                       // Move received data to output
                       #tempRet := INT_TO_WORD(MOVE_BLK_VARIANT(SRC := #statRcvBuffer,
                                                                                        COUNT := MIN(IN1 := #tempChunk.lenData, IN2 := #statSizeRcvArray - #statRcvdLen), // Move as much as possible to output
                                                                                        SRC_INDEX := #tempChunk.posData,
                                                                                        DEST_INDEX := UDINT_TO_DINT(#statRcvdLen),
                                                                                        DEST => #responseData));

                       // Exit loop immediately and output error if data could not be moved
                       IF #tempRet <> 0 THEN
                         #statStatusID := #STATUS_ID_MOVE_CHUNKED;
                         #statStatus := #tempRet;
                         EXIT;
                       END_IF;

                       // Move start position of data behind data of current chunk in case packet contains more data; only relevant if REPEAT loop is executed again
                       #tempChunk.posData += #tempChunk.lenData;

                       // Subtract length of data in current packet from remaining length of chunk and add to sum of received data
                       #statChunkLen -= #tempChunk.lenData;
                       #statRcvdLen += #tempChunk.lenData;

                       IF #statRcvdLen > #statSizeRcvArray THEN // Receive buffer too small
                         #statStatus := #STATUS_BUFFER_SIZE;
                         #statLength := #statRcvdLen; // Output required size of buffer according to so far received chunked messages
                       END_IF;
                     END_IF;
                   UNTIL (#tempChunk.exitLoop = true) END_REPEAT;
                 END_IF;
               END_REGION

             ELSIF #instTRcv.ERROR THEN
               #statStatusID := #STATUS_ID_TRCV;
               #statStatus := #instTRcv.STATUS;
             END_IF;
           END_REGION

         ELSE // Undefined state in state machine reached
           #statStatus := #STATUS_UNDEFINED_STATE;
       END_CASE;

     UNTIL (#tempExitLoop = true) END_REPEAT;
   END_REGION

   REGION OUTPUTS
     // Write outputs
     IF (#statStatus = #STATUS_DONE) AND (#statDone = false) THEN // Execution finished without errors
       #statDone := true;
       #statBusy := false;
       #statError := false;
       #statSend.connect := false;
       #statSend.req := false;
       #statTimeoutIn := false;
       #statFBState := #STATE_IDLE; // Switch state machine to "no processing"

     ELSIF (#statStatus.%X15 = true) AND (#statError = false) THEN // Error occurred (#statStatus is 16#8000 to 16#FFFF)
       #statDone := false;
       #statBusy := false;
       #statError := true;
       #statSend.connect := false;
       #statSend.req := false;
       #statTimeoutIn := false;
       #statFBState := #STATE_IDLE; // Switch state machine to "no processing"

     ELSIF (#execute = false) AND ((#statDone = true) OR (#statError = true)) THEN // Reset outputs
       #statDone := false;
       #statBusy := false;
       #statError := false;
       #statStatusID := 0;
       #statStatus := #STATUS_IDLE;
       #statResponseCode := 0;
       #statLength := 0;
       #statContentLength := 0;
       #statChunkLen := 0;
       #statEncoding := '';
       #statRcvdLen := 0;
       #statTimeoutIn := false;
     END_IF;

     // Write static values to outputs
     #done := #statDone;
     #busy := #statBusy;
     #error := #statError;
     #statusID := #statStatusID;
     #status := #statStatus;
     #responseCode := #statResponseCode;
     #length := #statLength;
   END_REGION OUTPUTS
END_FUNCTION_BLOCK

// folder: REST/Utilities

FUNCTION "LHTTP_ExtractStringFromArray" : Word   // FC2, SCL
{ S7_Optimized_Access := 'TRUE' }
VERSION : 0.1
   VAR_INPUT
      textBefore : String;   // Text before text that is extracted
      textAfter : String;   // Text after text that is extracted
   END_VAR
   VAR_OUTPUT
      extractedString : String;   // Extracted string
   END_VAR
   VAR_IN_OUT
      searchIn : Array[*] of Char;   // Array of Char to search in
   END_VAR
   VAR_TEMP
      tempLowerBound : DInt;   // Lower bound of given array
      tempNumElements : UDInt;   // Number of elements in given array
      tempPosInArray : DInt;   // Position in array during search
      tempLenTextBefore : Int;   // Length of text before
      tempPosTextBefore : DInt;   // Position of text before in array of Char
      tempLenTextAfter : Int;   // Length of text after
      tempPosTextAfter : Int;   // Position of text after in converted string
      tempString : String;   // Temporary string to work with
   END_VAR
   // Ret_Val : Return value; 16#0000: Successful, text was found, 16#9001: Unsuccessful, only start text was found, extracted String is filled with characters after start text, 16#9002: Unsuccessful, neither text was found
   VAR CONSTANT
      LEN_STRING : UInt := 254;   // Max. length of String
      STATUS_TEXT_FOUND : Word := 16#0000;   // Texts before and after were found
      STATUS_ONLY_START : Word := 16#9001;   // Only text before was found
      STATUS_NOTHING_FOUND : Word := 16#9002;   // Neither text was found
   END_VAR
BEGIN
   //=============================================================================
   // SIEMENS AG
   // (c)Copyright 2019
   //-----------------------------------------------------------------------------
   // Library:       LHTTP
   // Tested with:   CPU 1516-3 PN/DP V2.6
   // Engineering:   TIA Portal V15.1
   // Restrictions:  --
   // Requirements:  --
   // Functionality: Extracts a String specified by a text before and after
   //                from an array of Char
   //-----------------------------------------------------------------------------
   // Change log table:
   // Version    Date         Expert in charge         Changes applied
   // 01.00.00   01.04.2019   Siemens Online Support   First released version
   //=============================================================================

   // Initialization
   #tempPosTextBefore := 0;
   #tempPosTextAfter := 0;
   #tempLenTextBefore := LEN(#textBefore);
   #tempLenTextAfter := LEN(#textAfter);
   #extractedString := '';
   #LHTTP_ExtractStringFromArray := #STATUS_NOTHING_FOUND;

   // Get number of elements
   #tempPosInArray := #tempLowerBound := LOWER_BOUND(ARR := #searchIn, DIM := 1);
   #tempNumElements := DINT_TO_UDINT(UPPER_BOUND(ARR := #searchIn, DIM := 1) - #tempLowerBound + 1);


   // Search for text before until something was found
   REPEAT

     // Convert Chars to String
     Chars_TO_Strg(Chars  := #searchIn,
                   pChars := #tempPosInArray - #tempLowerBound, // Subtract offset since pChars is zero based
                   Cnt    := UDINT_TO_UINT(MIN(IN1 := #LEN_STRING, IN2 := #tempNumElements)),
                   Strg   => #tempString);

     // Search for text before
     #tempPosTextBefore := FIND(IN1 := #tempString, IN2 := #textBefore);

     // Text before was found
     IF #tempPosTextBefore > 0 THEN

       // Set position in array to end of text before
       #tempPosInArray += #tempPosTextBefore + #tempLenTextBefore - 1;

       // Create new string from end of text before
       Chars_TO_Strg(Chars  := #searchIn,
                     pChars := #tempPosInArray - #tempLowerBound, // Subtract offset since pChars is zero based
                     Cnt    := UDINT_TO_UINT(MIN(IN1 := #LEN_STRING, IN2 := #tempNumElements)),
                     Strg   => #tempString);

       // Find end of string to be extracted
       #tempPosTextAfter := FIND(IN1 := #tempString, IN2 := #textAfter);

       IF #tempPosTextAfter > 0 THEN // Shorten string if text after was found

         #extractedString := LEFT(IN := #tempString, L := #tempPosTextAfter - 1);
         #LHTTP_ExtractStringFromArray := #STATUS_TEXT_FOUND;
         EXIT;

       ELSE // Output whole string if text after was not found

         #extractedString := #tempString;
         #LHTTP_ExtractStringFromArray := #STATUS_ONLY_START;
         EXIT;

       END_IF;

     ELSE
       // Otherwise continue search in next string minus length of text before to ensure
       // keywords are not broken up at the end of a string and thus missed
       #tempPosInArray += UINT_TO_INT(#LEN_STRING) - #tempLenTextBefore;
     END_IF;

     // Repeat until end of array is reached
   UNTIL (#tempPosInArray > #tempNumElements) END_REPEAT;
END_FUNCTION

FUNCTION "LHTTP_FindStringInArray" : DInt   // FC5, SCL
{ S7_Optimized_Access := 'TRUE' }
VERSION : 0.1
   VAR_INPUT
      searchFor : String;   // Text that is searched for
   END_VAR
   VAR_IN_OUT
      searchIn : Array[*] of Char;   // Array of Char to search in
   END_VAR
   VAR_TEMP
      tempLowerBound : DInt;   // Lower bound of given array
      tempNumElements : UDInt;   // Number of elements in given array
      tempLenSearchFor : Int;   // Length of text that is seached for
      tempPosInArray : DInt;   // Position in array during search (0-based)
      tempPosInString : Int;   // Position in working string during search
      tempString : String;   // Temporary string to work with
   END_VAR
   // Ret_Val : Position (index) of the first character of the text that is searched for within the array of Char
   VAR CONSTANT
      LEN_STRING : UInt := 254;   // Max. length of String
   END_VAR
BEGIN
   //=============================================================================
   // SIEMENS AG
   // (c)Copyright 2019
   //-----------------------------------------------------------------------------
   // Library:       LHTTP
   // Tested with:   CPU 1516-3 PN/DP V2.6
   // Engineering:   TIA Portal V15.1
   // Restrictions:  --
   // Requirements:  --
   // Functionality: Searches for a specified String within an array of Char
   //-----------------------------------------------------------------------------
   // Change log table:
   // Version    Date         Expert in charge         Changes applied
   // 01.00.00   01.01.2019   Siemens Online Support   First released version
   //=============================================================================

   // Initialization
   #tempPosInString := 0;
   #tempPosInArray := 0;
   #tempLenSearchFor := LEN(#searchFor);
   #LHTTP_FindStringInArray := -1;

   // Get number of elements
   #tempLowerBound := LOWER_BOUND(ARR := #searchIn, DIM := 1);
   #tempNumElements := DINT_TO_UDINT(UPPER_BOUND(ARR := #searchIn, DIM := 1) - #tempLowerBound + 1);

   // Search for beginning of text until something was found
   REPEAT

     // Convert Chars to String
     Chars_TO_Strg(Chars := #searchIn,
                   pChars := #tempPosInArray,
                   Cnt := UDINT_TO_UINT(MIN(IN1 := #LEN_STRING, IN2 := #tempNumElements)),
                   Strg => #tempString);

     // Search for text at beginning
     #tempPosInString := FIND(IN1 := #tempString, IN2 := #searchFor);

     // Keyword was found
     IF #tempPosInString > 0 THEN
       // Output position of string
       #LHTTP_FindStringInArray := #tempLowerBound + #tempPosInArray + #tempPosInString - 1;
       EXIT;
     ELSE
       // Otherwise continue search in next string minus length of text at beginning to ensure
       // keywords are not broken up at the end of a string and thus missed
       #tempPosInArray += UINT_TO_INT(#LEN_STRING) - #tempLenSearchFor;
     END_IF;

   UNTIL (#tempPosInString > 0) OR (#tempPosInArray > #tempNumElements) END_REPEAT;
END_FUNCTION

// ===== library: MasterCopy "REST_Param" =====

// folder: REST

DATA_BLOCK "REST_Param"   // DB2
{ S7_Optimized_Access := 'TRUE' }
VERSION : 0.1
   VAR
      get : Struct
         conn : TCON_IP_v4;
         execute : Bool;
         url : String := 'http://192.168.0.124/api/v2.0.0/log/error_reports/13';
         data : String;
         done : Bool;
         busy : Bool;
         error : Bool;
         statusID : USInt;
         status : Word;
         responseCode : UInt;
         length : UDInt;
      END_STRUCT;
      post : Struct
         execute : Bool;
         conn : TCON_IP_v4;
         url : String := '192.168.0.124/api/v2.0.0/log/error_reports';
         data : String := '{"description": "Hello"}';
      END_STRUCT;
   END_VAR
BEGIN
   get.conn.RemotePort := 80;
   get.conn.RemoteAddress.ADDR[4] := 124;
   get.conn.RemoteAddress.ADDR[2] := 168;
   get.conn.RemoteAddress.ADDR[1] := 192;
   get.conn.ActiveEstablished := true;
   get.conn.ID := 16#01;
   get.conn.InterfaceId := 64;
   post.conn.InterfaceId := 64;
   post.conn.ID := 16#02;
   post.conn.ActiveEstablished := true;
   post.conn.RemoteAddress.ADDR[1] := 192;
   post.conn.RemoteAddress.ADDR[2] := 168;
   post.conn.RemoteAddress.ADDR[4] := 124;
   post.conn.RemotePort := 80;
END_DATA_BLOCK

// ===== library: MasterCopy "REST_Response" =====

// folder: REST

DATA_BLOCK "REST_Response"   // DB4
{ S7_Optimized_Access := 'TRUE' }
VERSION : 0.1
   VAR
      data : Array[0..6000] of Char;
   END_VAR
BEGIN
END_DATA_BLOCK